(* PLC project Untitled1, Beckhoff Automation GmbH TF6420 Database Server Query Analyser 1.0.0.0 *)
(* stored: creationDateTime 2016-04-18T15:14:22, modificationDateTime 2016-04-18T15:14:22 *)

TYPE ST_TEMP1_Save : STRUCT
  id : DINT;
  timestamp : DT;
  temp1 : STRING(45);
END_STRUCT;
END_TYPE
